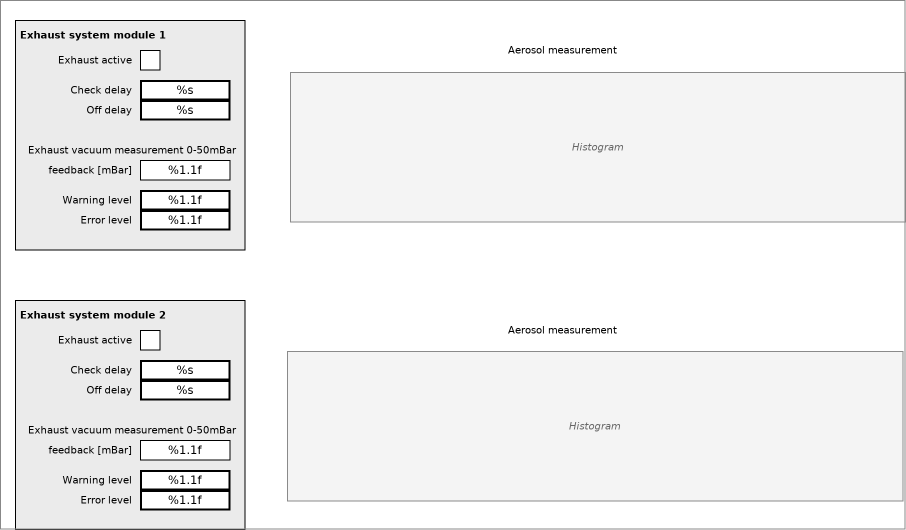
VISUALIZATION VISU_EXHAUST  // 906x530
    Rectangle (15,20 230x230)
    Rectangle (17,25 192x20), "Exhaust system module 1"
    Rectangle (45,80 90x20), "Check delay"
    Rectangle (140,80 90x20), "%s", text variable: PRG_MACHINE.fb_ExhaustSystem[1].tR_VacuumCheckDelay
        OnMouseDown: write the text variable via Edit
    Rectangle (45,100 90x20), "Off delay"
    Rectangle (140,100 90x20), "%s", text variable: PRG_MACHINE.fb_ExhaustSystem[1].tR_FUOffDelay
        OnMouseDown: write the text variable via Edit
    RoundedRectangle (140,50 20x20), colour toggle: PRG_MACHINE.fb_ExhaustSystem[1].bO_FUActivate
    Rectangle (35,50 100x20), "Exhaust active"
    Rectangle (25,140 220x20), "Exhaust vacuum measurement 0-50mBar"
    Rectangle (45,160 90x20), "feedback [mBar]"
    Rectangle (140,160 90x20), "%1.1f", text variable: PRG_MACHINE.fb_ExhaustSystem[1].fL_VacuumAnalogLevelMBar
    Histogram (290,72 616x150), scale format: %.1f, scale 0..2
        p1518820177: PRG_MACHINE.fb_ExhaustSystem[1].fL_ParticleMeasurements
        p102497268: PRG_MACHINE.fb_ExhaustSystem[1].fL_ParticleMeasurements
        p788070771: ARRAY [1..iC_ParticleMeasurementNb] OF REAL
    Rectangle (505,40 220x20), "Aerosol measurement"
    Rectangle (45,190 90x20), "Warning level"
    Rectangle (140,190 90x20), "%1.1f", text variable: PRG_MACHINE.fb_ExhaustSystem[1].fR_VacuumWarningLevelMBar
        OnMouseDown: write the text variable via Edit
    Rectangle (45,210 90x20), "Error level"
    Rectangle (140,210 90x20), "%1.1f", text variable: PRG_MACHINE.fb_ExhaustSystem[1].fR_VacuumErrorLevelMBar
        OnMouseDown: write the text variable via Edit
    Rectangle (15,300 230x230)
    Rectangle (17,305 192x20), "Exhaust system module 2"
    Rectangle (45,360 90x20), "Check delay"
    Rectangle (140,360 90x20), "%s", text variable: PRG_MACHINE.fb_ExhaustSystem[2].tR_VacuumCheckDelay
        OnMouseDown: write the text variable via Edit
    Rectangle (45,380 90x20), "Off delay"
    Rectangle (140,380 90x20), "%s", text variable: PRG_MACHINE.fb_ExhaustSystem[2].tR_FUOffDelay
        OnMouseDown: write the text variable via Edit
    RoundedRectangle (140,330 20x20), colour toggle: PRG_MACHINE.fb_ExhaustSystem[2].bO_FUActivate
    Rectangle (35,330 100x20), "Exhaust active"
    Rectangle (25,420 220x20), "Exhaust vacuum measurement 0-50mBar"
    Rectangle (45,440 90x20), "feedback [mBar]"
    Rectangle (140,440 90x20), "%1.1f", text variable: PRG_MACHINE.fb_ExhaustSystem[2].fL_VacuumAnalogLevelMBar
    Histogram (287,351 616x150), scale format: %.1f, scale 0..2
        p1518820177: PRG_MACHINE.fb_ExhaustSystem[2].fL_ParticleMeasurements
        p102497268: PRG_MACHINE.fb_ExhaustSystem[2].fL_ParticleMeasurements
        p788070771: ARRAY [1..iC_ParticleMeasurementNb] OF REAL
    Rectangle (505,320 220x20), "Aerosol measurement"
    Rectangle (45,470 90x20), "Warning level"
    Rectangle (140,470 90x20), "%1.1f", text variable: PRG_MACHINE.fb_ExhaustSystem[2].fR_VacuumWarningLevelMBar
        OnMouseDown: write the text variable via Edit
    Rectangle (45,490 90x20), "Error level"
    Rectangle (140,490 90x20), "%1.1f", text variable: PRG_MACHINE.fb_ExhaustSystem[2].fR_VacuumErrorLevelMBar
        OnMouseDown: write the text variable via Edit
END_VISUALIZATION

// ---- VISUs/Projects/Machine/VISU_CLEAN_PROCESS.TcVIS
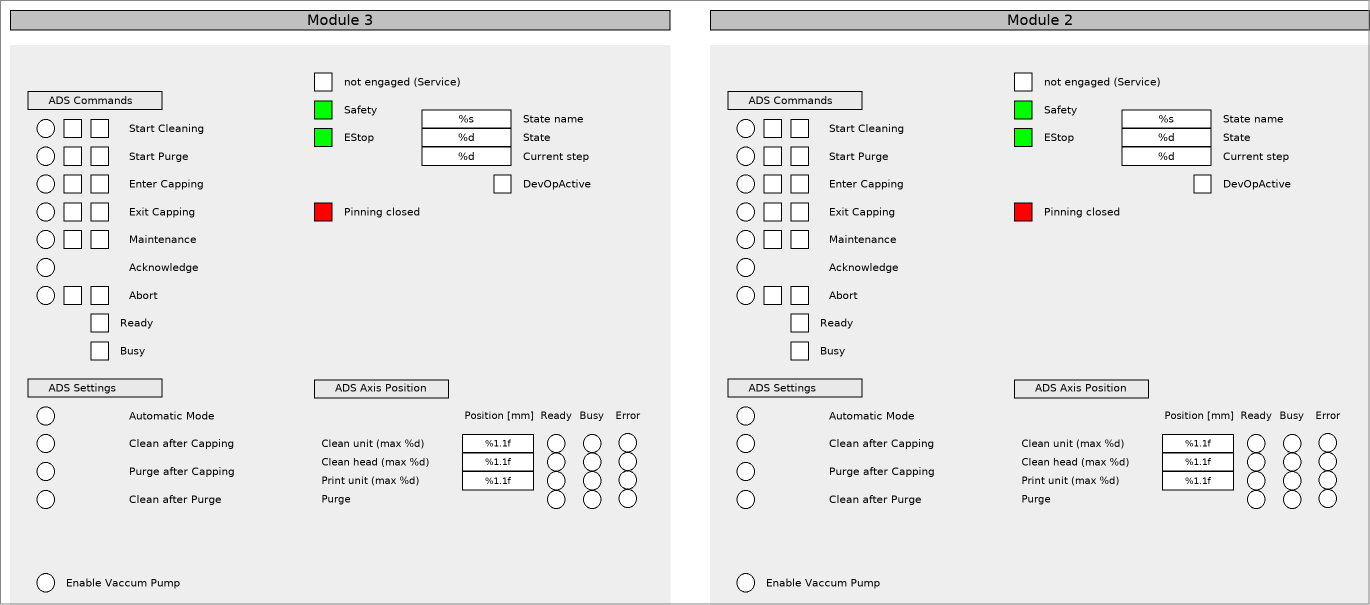
VISUALIZATION VISU_CLEAN_PROCESS  // 1370x605
    Frame (10,45 660x560)
        shows _VISU_CLEAN_PROCESS(m_Inst := 2)
    Rectangle (10,10 660x20), "Module 3"
    Rectangle (710,10 660x20), "Module 2"
    Frame (710,45 660x560)
        shows _VISU_CLEAN_PROCESS(m_Inst := 1)
END_VISUALIZATION

// ---- VISUs/Projects/Machine/VISU_CLEAN_PU.TcVIS
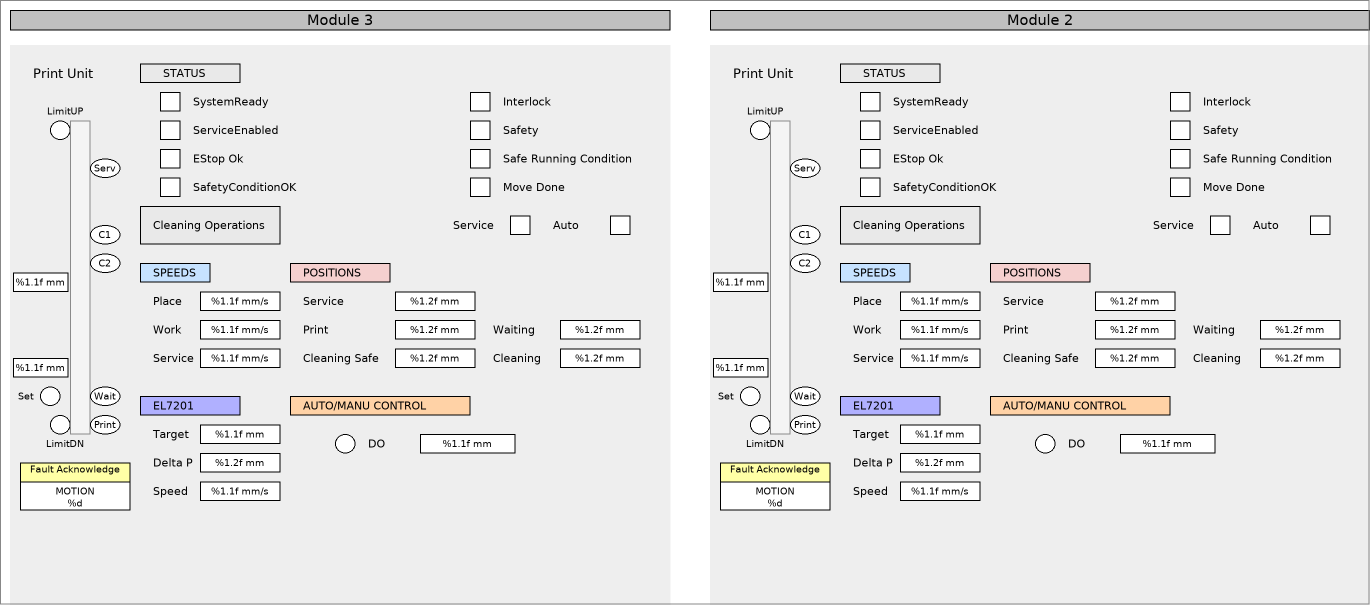
VISUALIZATION VISU_CLEAN_PU  // 1370x605
    Frame (10,45 660x560)
        shows _VISU_CLEAN_PU(m_Inst := 2)
    Rectangle (10,10 660x20), "Module 3"
    Rectangle (710,10 660x20), "Module 2"
    Frame (710,45 660x560)
        shows _VISU_CLEAN_PU(m_Inst := 1)
END_VISUALIZATION

// ---- VISUs/Projects/Machine/VISU_MACHINE.TcVIS
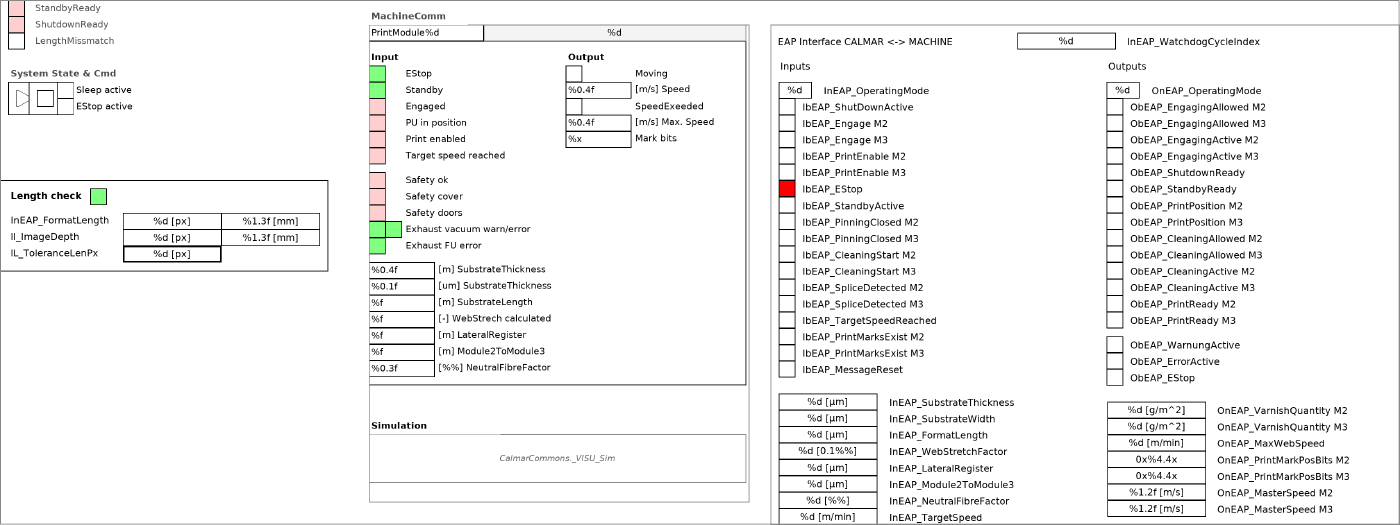
VISUALIZATION VISU_MACHINE  // 1708x641
    Frame (450,30 464x583)
        shows _VISU_MachineComm(mInst := PRG_MACHINE.fbMachineComm)
    Rectangle (450,10 120x20), "MachineComm"
    Rectangle (0,220 400x111)
    Rectangle (270,260 120x20), "%1.3f [mm]", text variable: PRG_MACHINE.InEAP_FormatLength / 1000
    Rectangle (10,260 136x18), "InEAP_FormatLength"
    Rectangle (10,230 96x18), "Length check"
    Rectangle (150,260 120x20), "%d [px]", text variable: PRG_MACHINE.lL_SubstrateLenPx
    Rectangle (270,280 120x20), "%1.3f [mm]", text variable: PRG_PRINT.sAdsPrintUnit[ePr_PU_UNIT_1].sI_JobSettings.lI_ImageDepth / 1000
    Rectangle (10,280 136x18), "lI_ImageDepth"
    Rectangle (150,280 120x20), "%d [px]", text variable: PRG_MACHINE.lL_ImageDepthPx
    RoundedRectangle (110,230 20x20), colour toggle: PRG_MACHINE.bL_MismatchLength
    Rectangle (10,300 136x18), "lL_ToleranceLenPx"
    Rectangle (150,300 120x20), "%d [px]", text variable: PRG_MACHINE.lL_ToleranceLenPx
        OnMouseClick: write the text variable via Default
    Frame (940,30 768x611)
        shows VISU_EAP_MACHINE()
    RoundedRectangle (10,0 20x20)
        toggle PRG_MACHINE.ObEAP_StandbyReady
    Rectangle (40,0 140x20), "StandbyReady"
    RoundedRectangle (10,20 20x20)
        toggle PRG_MACHINE.ObEAP_ShutdownReady
    Rectangle (40,20 140x20), "ShutdownReady"
    RoundedRectangle (10,40 20x20)
        toggle PRG_MACHINE.ObEAP_ShutdownReady
    Rectangle (40,40 140x20), "LengthMissmatch"
    Rectangle (10,80 160x20), "System State & Cmd"
    Group (10,100 20x20), input disabled if: NOT PRG_MACHINE.sADS_Machine[1].sI_Sleep.bO_CommandCanEx
        tap PRG_MACHINE.bL_SleepVisu
        RoundedRectangle (0,0 40x40)
        Polygon (10,10) (12,10) (30,20) (12,30) (10,30)
    Group (35,100 20x20), input disabled if: NOT PRG_MACHINE.sADS_Machine[1].sI_WakeUp.bO_CommandCanEx
        tap PRG_MACHINE.bL_WakeUpVisu
        RoundedRectangle (0,0 40x40)
        Rectangle (10,10 20x20)
    RoundedRectangle (70,100 20x20), colour toggle: PRG_MACHINE.sO_SystemCmd.bSleep
    RoundedRectangle (70,120 20x20), colour toggle: PRG_MACHINE.sO_SystemCmd.bEStop
    RoundedRectangle (90,100 100x20), "Sleep active"
    RoundedRectangle (90,120 100x20), "EStop active"
END_VISUALIZATION

// ---- VISUs/Projects/Print/VISU_ButtonBack.TcVIS
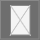
VISUALIZATION VISU_ButtonBack  // 40x40
    RoundedRectangle (0,0 40x40)
        OnMouseClick: change screen: Previous 
    Image (10,5 20x30), image: arrow-return-left_w
        OnMouseClick: change screen: Previous 
END_VISUALIZATION

// ---- VISUs/Projects/Print/VISU_Cameras.TcVIS
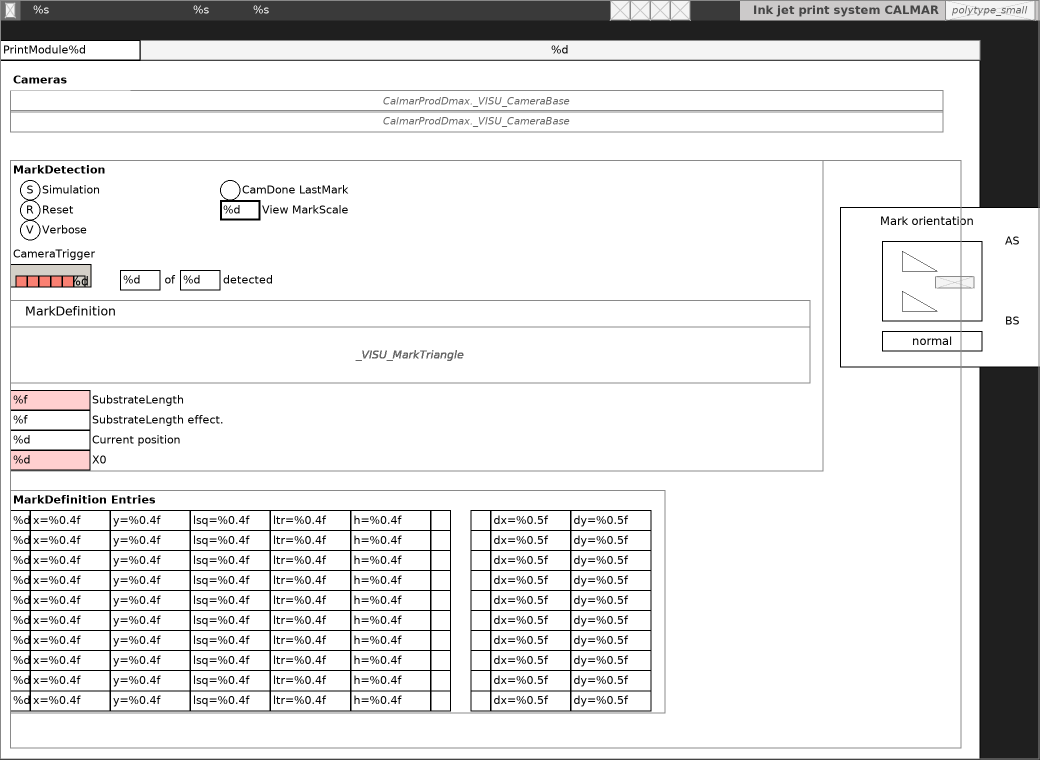
VISUALIZATION VISU_Cameras  // 1040x760
    Rectangle (0,60 980x700)
    Frame (10,160 951x588)
        shows _VISU_MarkCamera_WEU(mCam := PRG_PRINT.fbPrintModule[PRG_PRINT.fbModuleMaster.nViewPmSel].fbMarkCameraWeu, mMarkDetect := PRG_PRINT.fbPrintModule[PRG_PRINT.fbModuleMaster.nViewPmSel].fbMarkDetection)
    Frame (10,90 933x22)
        shows CalmarProdDmax._VISU_CameraBase(m_Inst := PRG_PRINT.fbPrintModule[PRG_PRINT.fbModuleMaster.nViewPmSel].fbNoCamera)
    Frame (10,110 933x22)
        shows CalmarProdDmax._VISU_CameraBase(m_Inst := PRG_PRINT.fbPrintModule[PRG_PRINT.fbModuleMaster.nViewPmSel].fbMarkCameraWeu)
    Scrollbar (140,40 840x20), "%d", text variable: PRG_PRINT.fbModuleMaster.nViewPmSel
        p1057716461: PRG_PRINT.fbModuleMaster.nViewPmSel
    Rectangle (0,40 140x20), "PrintModule%d", text variable: PRG_PRINT.fbModuleMaster.nViewPmSel
    Frame (20,0 1020x20)
        shows VISU_Header()
    Frame (0,0 20x20)
        shows VISU_ButtonBack()
    Rectangle (10,70 120x20), "Cameras"
END_VISUALIZATION

// ---- VISUs/Projects/Print/VISU_Header.TcVIS
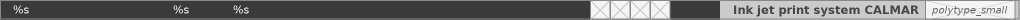
VISUALIZATION VISU_Header  // 1020x20
    Rectangle (0,0 1020x20)
    Rectangle (10,0 160x20), "%s", text variable: PRG_SYSTEM.sC_Ads_System.aProject
    Rectangle (170,0 60x20), "%s", text variable: PRG_SYSTEM.sC_Ads_System.aMachine
    Rectangle (230,0 120x20), "%s", text variable: PRG_SYSTEM.aCurrentDateTime
    Image (650,0 20x20), invisible if: NOT PRG_MACHINE.bO_ErrorMsgActive, image: GlobalImagePool.error_icon
    Image (610,0 20x20), invisible if: NOT PRG_MACHINE.sO_SystemCmd.bEStop, image: GlobalImagePool.estop_icon
    Image (590,0 20x20), invisible if: NOT PRG_MACHINE.sO_SystemCmd.bSleep, image: GlobalImagePool.sleep_icon
    Image (630,0 20x20), invisible if: NOT PRG_MACHINE.bO_WarningMsgActive, image: GlobalImagePool.warning_icon
    Rectangle (720,0 300x20)
    Image (925,0 90x20), image: polytype_small
    Rectangle (730,0 200x20), "Ink jet print system CALMAR"
END_VISUALIZATION

// ---- VISUs/Projects/Print/VISU_ButtonHome.TcVIS
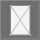
VISUALIZATION VISU_ButtonHome  // 40x40
    RoundedRectangle (0,0 40x40)
        OnMouseClick: change screen: VISU_Main
    Image (10,5 20x30), image: house_w
        OnMouseClick: change screen: VISU_Main
END_VISUALIZATION

// ---- VISUs/Projects/Print/VISU_PRINT.TcVIS
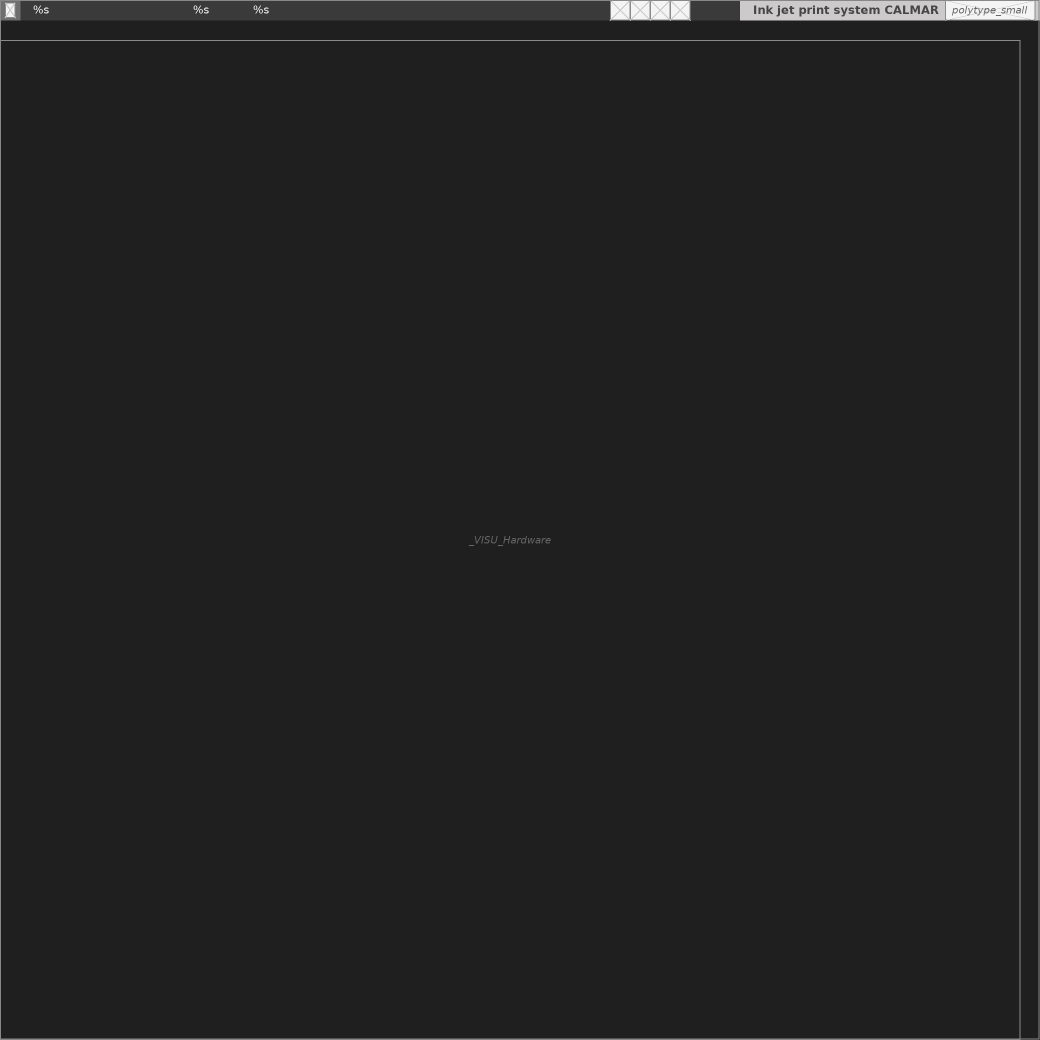
VISUALIZATION VISU_PRINT  // 1040x1040
    Frame (20,0 1020x20)
        shows VISU_Header()
    TabControl (0,40 1020x1000)
        shows _VISU_Hardware(m_fbHw := PRG_PRINT.fbHardwarePool)
        shows CalmarCompPrint._VISU_PU(m_Inst_Fb := PRG_PRINT.FB_PU[1])
        [0]: TabTitle=Hardware
    Frame (0,0 20x20)
        shows VISU_ButtonBack()
END_VISUALIZATION

// ---- VISUs/Projects/Print/VISU_PrintModule_Detail.TcVIS
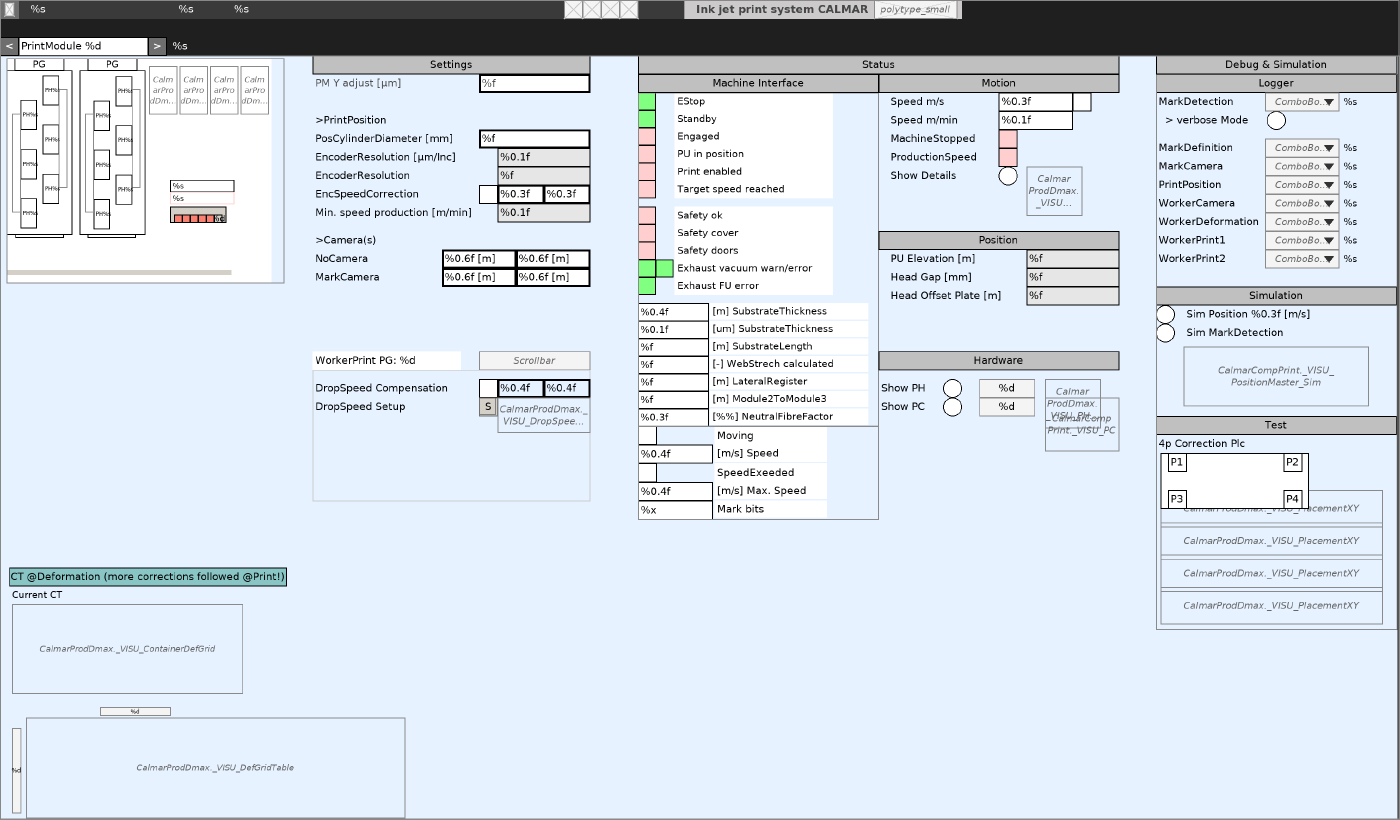
VISUALIZATION VISU_PrintModule_Detail  // 1514x887
    Rectangle (20,40 140x20), "PrintModule %d", text variable: PRG_PRINT.fbModuleMaster.nViewPmSel
    Frame (0,60 1514x827)
        shows _VISU_Pm_WEU(mInst := PRG_PRINT.fbPrintModule[PRG_PRINT.fbModuleMaster.nViewPmSel])
    Frame (20,0 1020x20)
        shows VISU_Header()
    Frame (0,0 20x20)
        shows VISU_ButtonBack()
    RoundedRectangle (160,40 20x20), ">"
        OnMouseClick: execute { PRG_PRINT.fbModuleMaster.nViewPmSel := PRG_PRINT.fbModuleMaster.nViewPmSel + 1; }
    RoundedRectangle (0,40 20x20), "<"
        OnMouseClick: execute { PRG_PRINT.fbModuleMaster.nViewPmSel := PRG_PRINT.fbModuleMaster.nViewPmSel - 1; }
    Rectangle (180,40 300x20), "%s", text variable: PRG_PRINT.fbModuleMaster._sModules[PRG_PRINT.fbModuleMaster.nViewPmSel]^._instanceName
END_VISUALIZATION

// ---- VISUs/Projects/Print/VISU_PrintOverview.TcVIS
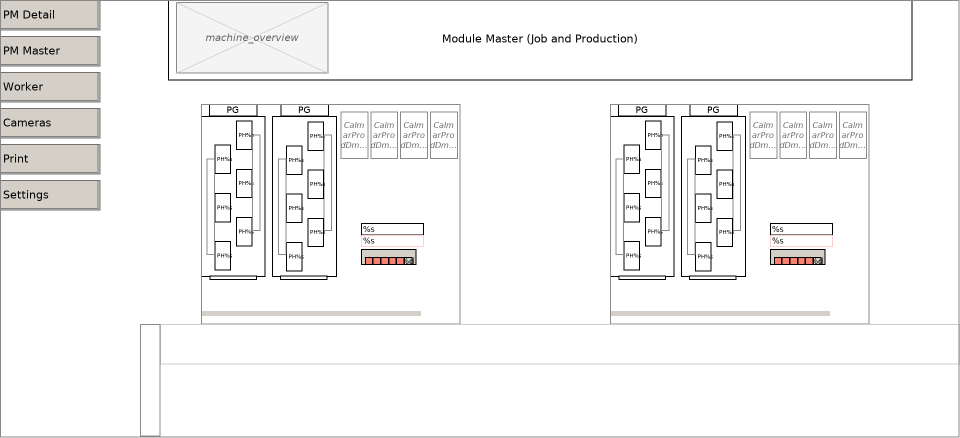
VISUALIZATION VISU_PrintOverview  // 960x438
    Button (0,144 100x30), "Print"
        OnMouseClick: change screen: VISU_PRINT
    Button (0,0 100x30), "PM Detail"
        OnMouseClick: change screen: VISU_PrintModule_Detail
    Button (0,72 100x30), "Worker"
        OnMouseClick: change screen: VISU_Workers
    Frame (610,104 259x220)
        shows _VISU_Pm_WEU_mini(mInst := PRG_PRINT.fbPrintModule[1])
    Frame (201,104 259x220)
        shows _VISU_Pm_WEU_mini(mInst := PRG_PRINT.fbPrintModule[2])
    Rectangle (160,324 800x40), colour toggle: PRG_PRINT.fbPrintOverview.bMovingInd
    Frame (140,324 20x112)
        shows CalmarProdDmax._VISU_CTsFlow(m_Inst := PRG_PRINT.fbPrintOverview)
    RoundedRectangle (168,-2 744x82), "Module Master (Job and Production)"
    Image (176,2 152x71), image: machine_overview
    Button (0,180 100x30), "Settings", input disabled if: TRUE
        OnMouseClick: change screen: VISU_SettingsWeu
    Button (0,108 100x30), "Cameras"
        OnMouseClick: change screen: VISU_Cameras
    Button (0,36 100x30), "PM Master", input disabled if: TRUE
        OnMouseClick: change screen: VISU_ModuleMaster
END_VISUALIZATION

// ---- VISUs/Projects/Print/VISU_Workers.TcVIS
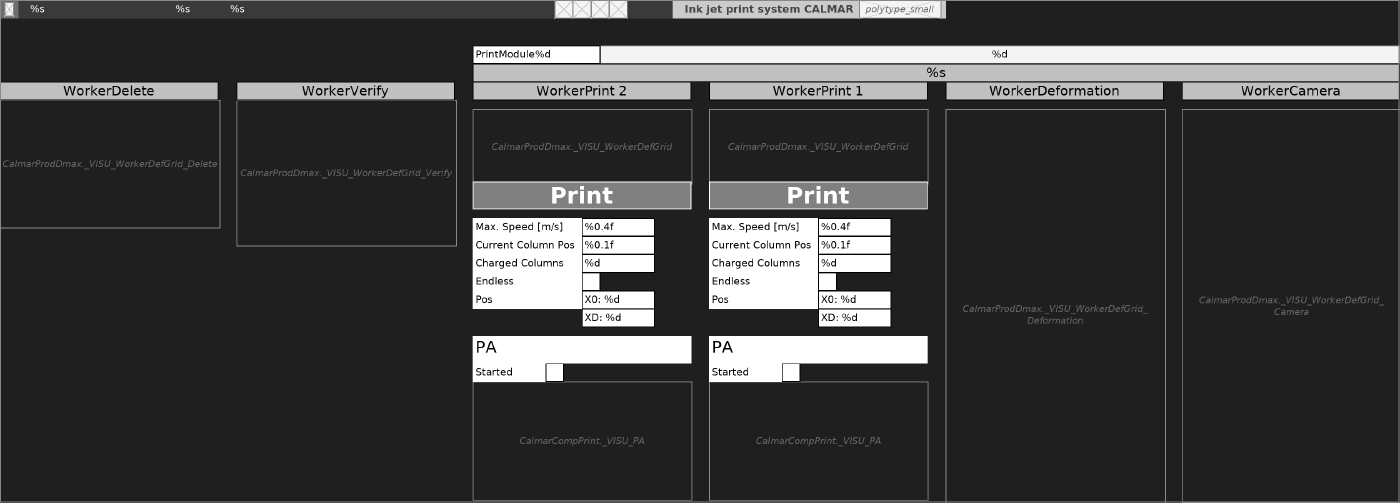
VISUALIZATION VISU_Workers  // 1540x554
    Frame (20,0 800x21)
        shows VISU_Header()
    Scrollbar (660,50 880x20), "%d", text variable: PRG_PRINT.fbModuleMaster.nViewPmSel
        p1057716461: PRG_PRINT.nSelectPmView
    Rectangle (520,50 140x20), "PrintModule%d", text variable: PRG_PRINT.fbModuleMaster.nViewPmSel
    Frame (520,70 762x484)
        shows _VISU_Pm_Worker(mInst := PRG_PRINT.fbPrintModule[PRG_PRINT.fbModuleMaster.nViewPmSel])
    Frame (0,110 242x141)
        shows CalmarProdDmax._VISU_WorkerDefGrid_Delete(m_Inst := PRG_PRINT.fbWorkerDelete)
    Frame (260,110 242x161)
        shows CalmarProdDmax._VISU_WorkerDefGrid_Verify(m_Inst := PRG_PRINT.fbWorkerVerify)
    Rectangle (0,90 240x20), "WorkerDelete"
    Rectangle (260,90 240x20), "WorkerVerify"
    Frame (0,0 20x20)
        shows VISU_ButtonBack()
END_VISUALIZATION

// ---- VISUs/Projects/Print/VIUS_TestnDebug.TcVIS
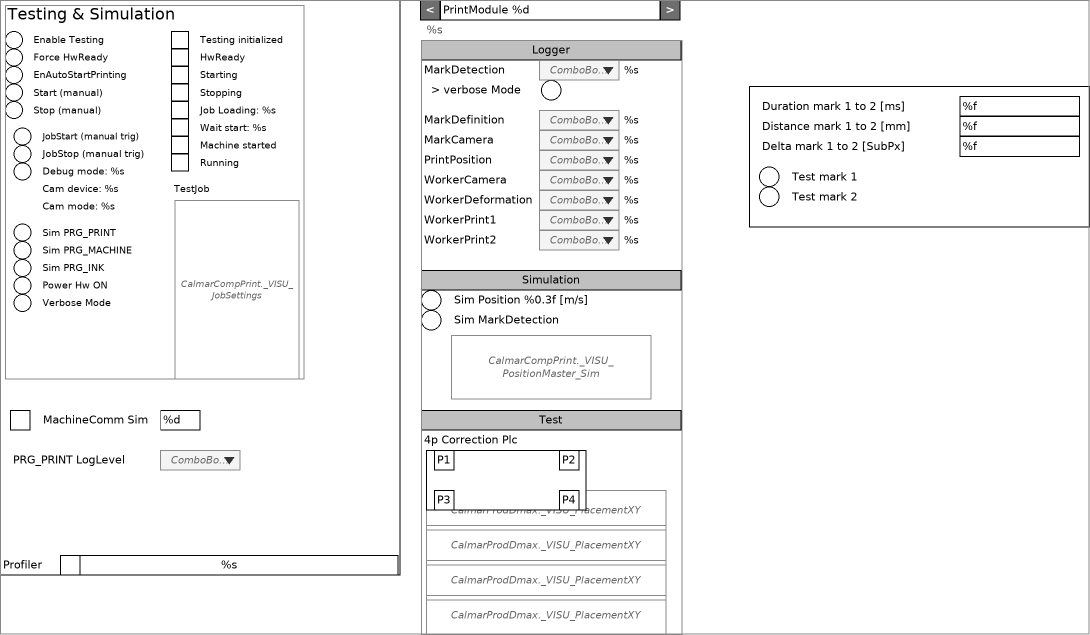
VISUALIZATION VIUS_TestnDebug  // 1090x635
    Rectangle (0,0 400x575)
    Frame (5,5 299x374)
        shows _VISU_PrgPrint_test(mInst := PRG_PRINT.fbPrgPrintTest)
    Rectangle (160,410 40x20), "%d", tooltip "Simulation mode", text variable: PRG_MACHINE.fbMachineComm._nModeSel
        OnMouseClick: write the text variable via Default
    Rectangle (40,410 120x20), "MachineComm Sim"
    RoundedRectangle (10,410 20x20)
        toggle PRG_MACHINE.fbMachineComm.bSimEnable
    Rectangle (10,450 140x20), "PRG_PRINT LogLevel"
    ComboBoxInteger (160,450 80x20), tooltip "LogLevel", variable: PRG_PRINT.ePrint_LogLevel, text list: 'LogSeverity'
    Rectangle (60,555 338x20), "%s", text variable: PRG_PRINT.fbProfiler.aProfilerData
    Rectangle (60,555 20x20)
        tap PRG_PRINT.fbProfiler.bReset
    Rectangle (0,555 60x20), "Profiler"
    RoundedRectangle (420,0 20x20), "<"
        OnMouseClick: execute { PRG_PRINT.fbModuleMaster.nViewPmSel := PRG_PRINT.fbModuleMaster.nViewPmSel - 1; }
    Rectangle (440,0 220x20), "PrintModule %d", text variable: PRG_PRINT.fbModuleMaster.nViewPmSel
    RoundedRectangle (660,0 20x20), ">"
        OnMouseClick: execute { PRG_PRINT.fbModuleMaster.nViewPmSel := PRG_PRINT.fbModuleMaster.nViewPmSel + 1; }
    Rectangle (420,20 260x20), "%s", text variable: PRG_PRINT.fbModuleMaster._sModules[PRG_PRINT.fbModuleMaster.nViewPmSel]^._instanceName
    Frame (421,40 261x595)
        shows _VISU_Pm_Debug(mInst := PRG_PRINT.fbPrintModule[1])
    Frame (749,86 341x141)
        shows _VISU_NeutralFiberDetermine(mInst := PRG_PRINT.fbNeutralFibreDetermine)
END_VISUALIZATION

// ---- VISUs/Projects/Print/_VISU_ButtonFrameSel.TcVIS
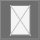
VISUALIZATION _VISU_ButtonFrameSel  // 40x40
VAR_IN_OUT
  mCfg : ST_ButtonFrameSel_Def;
END_VAR
    RoundedRectangle (0,0 40x40), tooltip "%s", colour toggle: mCfg.pFrameSelect^ = mCfg.nFrameIdx
        p4168582468: mCfg.sVisuName
        OnMouseClick: execute { mCfg.pFrameSelect^ := mCfg.nFrameIdx; }
    Image (10,5 20x30), tooltip "%s"
        p84334746: mCfg.sImgId
        p4168582468: mCfg.sVisuName
        OnMouseClick: execute { mCfg.pFrameSelect^ := mCfg.nFrameIdx; }
END_VISUALIZATION

// ---- VISUs/Projects/System/VISU_SERVICE.TcVIS
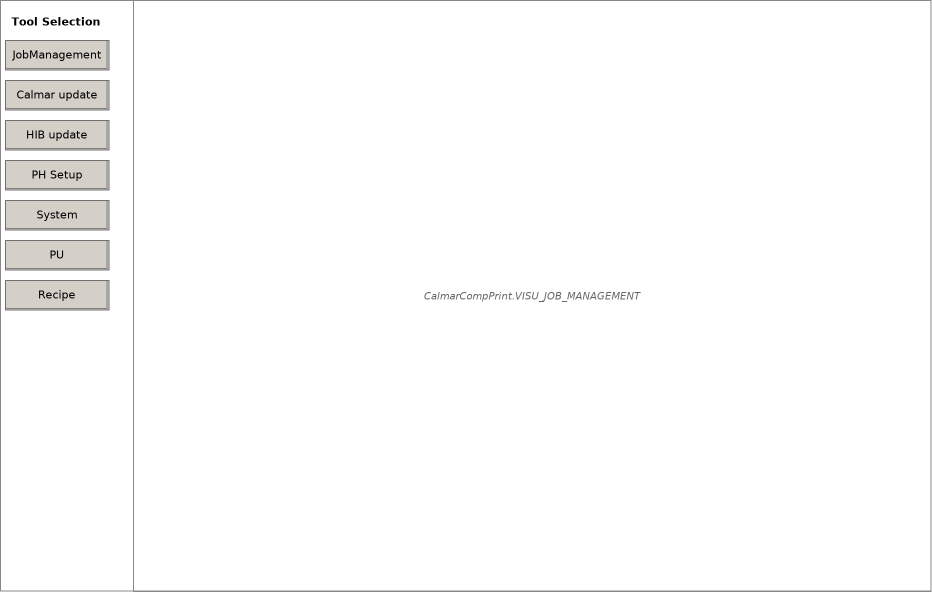
VISUALIZATION VISU_SERVICE  // 932x592
    Rectangle (0,0 932x592)
    Button (5,80 104x30), "Calmar update", colour toggle: PRG_PRINT.nServiceVisuFrameIndex = 1
        OnMouseClick: execute { PRG_PRINT.nServiceVisuFrameIndex := 1; }
    Button (5,40 104x30), "JobManagement", colour toggle: PRG_PRINT.nServiceVisuFrameIndex = 0
        OnMouseClick: execute { PRG_PRINT.nServiceVisuFrameIndex := 0; }
    Button (5,120 104x30), "HIB update", colour toggle: PRG_PRINT.nServiceVisuFrameIndex = 2
        OnMouseClick: execute { PRG_PRINT.nServiceVisuFrameIndex := 2; }
    Button (5,160 104x30), "PH Setup", colour toggle: PRG_PRINT.nServiceVisuFrameIndex = 3
        OnMouseClick: execute { PRG_PRINT.nServiceVisuFrameIndex := 3; }
    Button (5,200 104x30), "System", colour toggle: PRG_PRINT.nServiceVisuFrameIndex = 4
        OnMouseClick: execute { PRG_PRINT.nServiceVisuFrameIndex := 4; }
    Rectangle (4,7 104x30), "Tool Selection"
    Frame (133,0 798x592), frame switch variable: PRG_PRINT.nServiceVisuFrameIndex
        shows CalmarCompPrint.VISU_JOB_MANAGEMENT(m_Fb_JobManagement := PRG_PRINT.fbPrgPrintTest.fb_JobManagement)
        shows CalmarCompPrint.VISU_SETUP_CALMAR(m_fb_calmar_upd := PRG_PRINT.fbHardwarePool.fb_fwhw_update)
        shows CalmarCompPrint.VISU_SETUP_HIB(m_visu_fb := PRG_PRINT.fbHardwarePool.fb_hib_rup)
        shows CalmarCompPrint.VISU_SETUP_PH(m_Inst_fb_wave := PRG_PRINT.fb_fdl_waveform, m_Inst_fb_mask := PRG_PRINT.fb_fdl_mask)
        shows VISU_SYSTEM()
        shows CalmarCompPrint._VISU_PU(m_Inst_Fb := PRG_PRINT.FB_PU[1])
        shows CalmarCompSystem.VISU_RECIPE()
        [6]: m_visu_fb=PRG_PRINT.fb_visu_pu
        p2546873765: PRG_PRINT.fb_fdl_imgmap
        p2204176931: PRG_PRINT.fb_visu_pu
    Button (5,240 104x30), "PU", colour toggle: PRG_PRINT.nServiceVisuFrameIndex = 5
        OnMouseClick: execute { PRG_PRINT.nServiceVisuFrameIndex := 5; }
    Button (5,280 104x30), "Recipe", colour toggle: PRG_PRINT.nServiceVisuFrameIndex = 6
        OnMouseClick: execute { PRG_PRINT.nServiceVisuFrameIndex := 6; }
END_VISUALIZATION

// ---- VISUs/Projects/System/VISU_SYSTEM.TcVIS
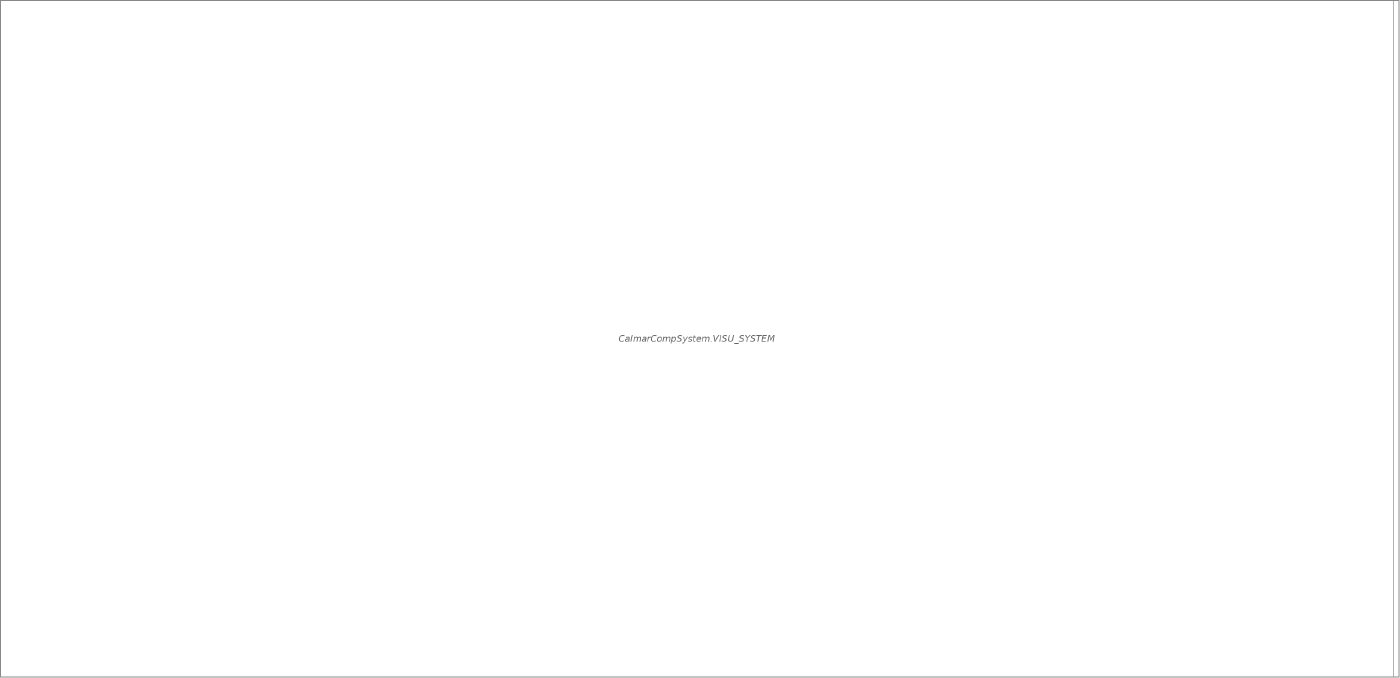
VISUALIZATION VISU_SYSTEM  // 1554x753
    Rectangle (0,0 1554x753)
    Frame (0,0 1547x752)
        shows CalmarCompSystem.VISU_SYSTEM()
END_VISUALIZATION

// ---- VISUs/Projects/VISU_INKSYSTEM.TcVIS
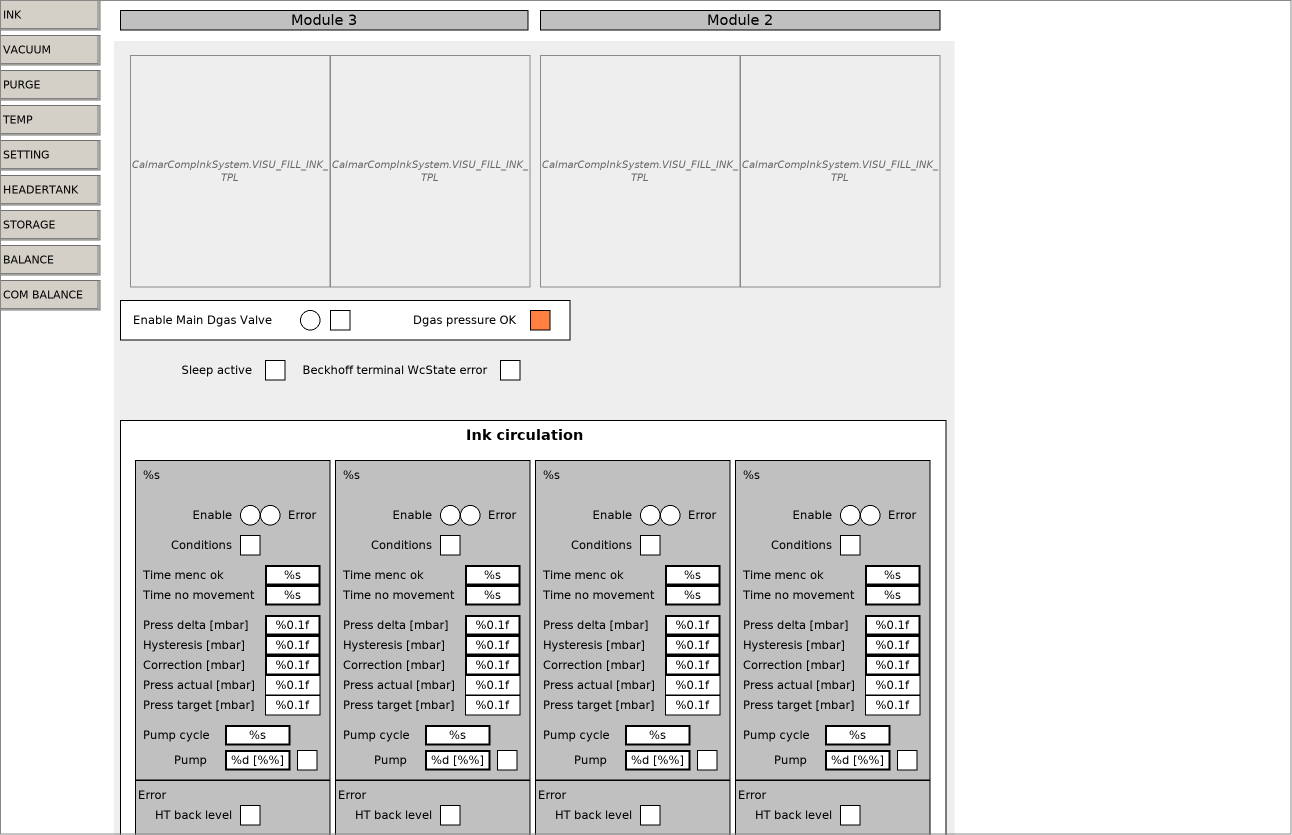
VISUALIZATION VISU_INKSYSTEM  // 1292x835
    Frame (110,0 1182x835), frame switch variable: PRG_INK.aVisuInkSystemFrameIndex
        shows VISU_INK()
        shows VISU_VACUUM()
        shows VISU_PURGE()
        shows VISU_TEMPERATUR()
        shows VISU_SETTINGS()
        shows VISU_HEADERTANK()
        shows VISU_ADS_INKSTORAGE_TANK_DVT()
        shows VISU_BALANCE()
        shows VISU_COMM_BALANCE()
    Button (0,0 100x30), "INK", colour toggle: PRG_INK.aVisuInkSystemFrameIndex = 0
        OnMouseClick: execute { PRG_INK.aVisuInkSystemFrameIndex := 0; }
    Button (0,70 100x30), "PURGE", colour toggle: PRG_INK.aVisuInkSystemFrameIndex = 2
        OnMouseClick: execute { PRG_INK.aVisuInkSystemFrameIndex := 2; }
    Button (0,105 100x30), "TEMP", colour toggle: PRG_INK.aVisuInkSystemFrameIndex = 3
        OnMouseClick: execute { PRG_INK.aVisuInkSystemFrameIndex := 3; }
    Button (0,140 100x30), "SETTING", colour toggle: PRG_INK.aVisuInkSystemFrameIndex = 4
        OnMouseClick: execute { PRG_INK.aVisuInkSystemFrameIndex := 4; }
    Button (0,210 100x30), "STORAGE", colour toggle: PRG_INK.aVisuInkSystemFrameIndex = 6
        OnMouseClick: execute { PRG_INK.aVisuInkSystemFrameIndex := 6; }
    Button (0,35 100x30), "VACUUM", colour toggle: PRG_INK.aVisuInkSystemFrameIndex = 1
        OnMouseClick: execute { PRG_INK.aVisuInkSystemFrameIndex := 1; }
    Button (0,175 100x30), "HEADERTANK", colour toggle: PRG_INK.aVisuInkSystemFrameIndex = 5
        OnMouseClick: execute { PRG_INK.aVisuInkSystemFrameIndex := 5; }
    Button (0,245 100x30), "BALANCE", colour toggle: PRG_INK.aVisuInkSystemFrameIndex = 7
        OnMouseClick: execute { PRG_INK.aVisuInkSystemFrameIndex := 7; }
    Button (0,280 100x30), "COM BALANCE", colour toggle: PRG_INK.aVisuInkSystemFrameIndex = 8
        OnMouseClick: execute { PRG_INK.aVisuInkSystemFrameIndex := 8; }
END_VISUALIZATION

// ---- VISUs/Projects/VISU_Main.TcVIS
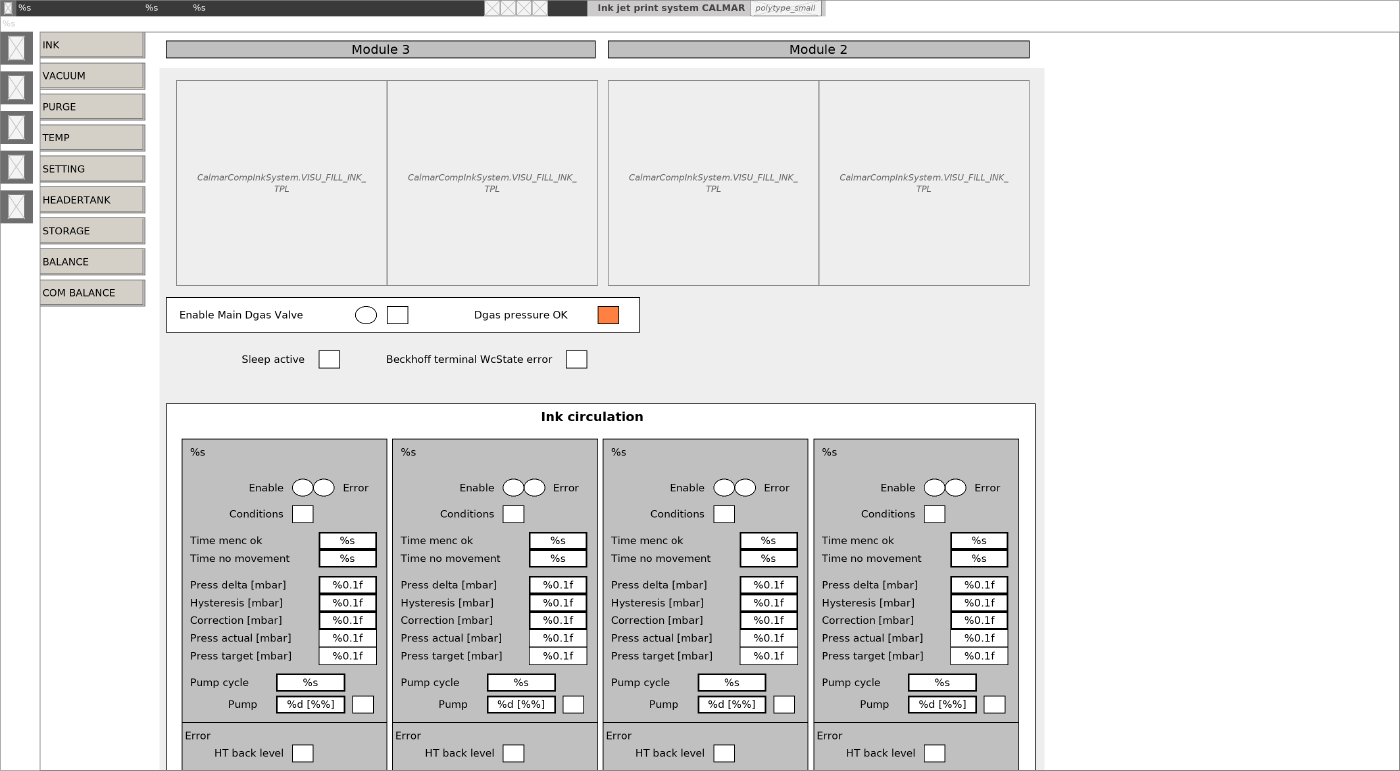
VISUALIZATION VISU_Main  // 1764x972
    Frame (50,40 1714x932), frame switch variable: PRG_SYSTEM.nMainVisuFrameIndex
        shows VISU_INKSYSTEM()
        shows VISU_PrintOverview()
        shows CalmarCompSystem.VISU_RECIPE()
        shows VISU_SERVICE()
        shows VISU_MACHINE()
    Frame (0,40 41x41)
        shows _VISU_ButtonFrameSel(mCfg := PRG_SYSTEM.sMainButtons[0])
    Rectangle (0,20 200x20), "%s", text variable: PRG_SYSTEM.sMainButtons[PRG_SYSTEM.nMainVisuFrameIndex].sVisuName
    Group (20,0 1020x20)
        Rectangle (0,0 1020x20)
        Rectangle (0,0 160x20), "%s", text variable: PRG_SYSTEM.sC_Ads_System.aProject
        Rectangle (160,0 60x20), "%s", text variable: PRG_SYSTEM.sC_Ads_System.aMachine
        Rectangle (220,0 120x20), "%s", text variable: PRG_SYSTEM.aCurrentDateTime
        Image (650,0 20x20), invisible if: NOT PRG_MACHINE.bO_ErrorMsgActive, image: GlobalImagePool.error_icon
        Image (610,0 20x20), invisible if: NOT PRG_MACHINE.sO_SystemCmd.bEStop, image: GlobalImagePool.estop_icon
        Image (590,0 20x20), invisible if: NOT PRG_MACHINE.sO_SystemCmd.bSleep, image: GlobalImagePool.sleep_icon
        Image (630,0 20x20), invisible if: NOT PRG_MACHINE.bO_WarningMsgActive, image: GlobalImagePool.warning_icon
        Rectangle (720,0 300x20)
        Image (925,0 90x20), image: polytype_small
        Rectangle (730,0 200x20), "Ink jet print system CALMAR"
    Frame (0,90 41x41)
        shows _VISU_ButtonFrameSel(mCfg := PRG_SYSTEM.sMainButtons[1])
    Frame (0,140 41x41)
        shows _VISU_ButtonFrameSel(mCfg := PRG_SYSTEM.sMainButtons[2])
    Frame (0,190 41x41)
        shows _VISU_ButtonFrameSel(mCfg := PRG_SYSTEM.sMainButtons[3])
    Frame (0,0 20x20)
        shows VISU_ButtonHome()
    Frame (0,240 41x41)
        shows _VISU_ButtonFrameSel(mCfg := PRG_SYSTEM.sMainButtons[4])
END_VISUALIZATION
